SUBAPPLICATION Uebung_080e2_AX (* Beispiel für E_CTU mit Eventbremse durch AX_D_FF / AUI_D_FF_TMIN *)
  (* Standard: 61499-2; Description: Copyright (c) 2023 Meisterschulen am Ostbahnhof This program and the accompanying materials are made available under the terms of the Eclipse Public License 2.0 which is available at https://www.eclipse.org/legal/epl-2.0/ SPDX-License-Identifier: EPL-2.0 *)
  (* Version 1.1, 2026-05-15, Franz Höpfinger, Meisterschulen am Ostbahnhof, Ported to AX Welt *)
  PACKAGE Uebungen;
  IMPORT logiBUS::io::DI::logiBUS_DI::Input_I1;
  IMPORT logiBUS::io::DI::logiBUS_DI::Input_I2;
  IMPORT logiBUS::io::DQ::logiBUS_DO::Output_Q1;
  IMPORT Uebungen::const::UT::DefaultPool::OutputNumber_N1;
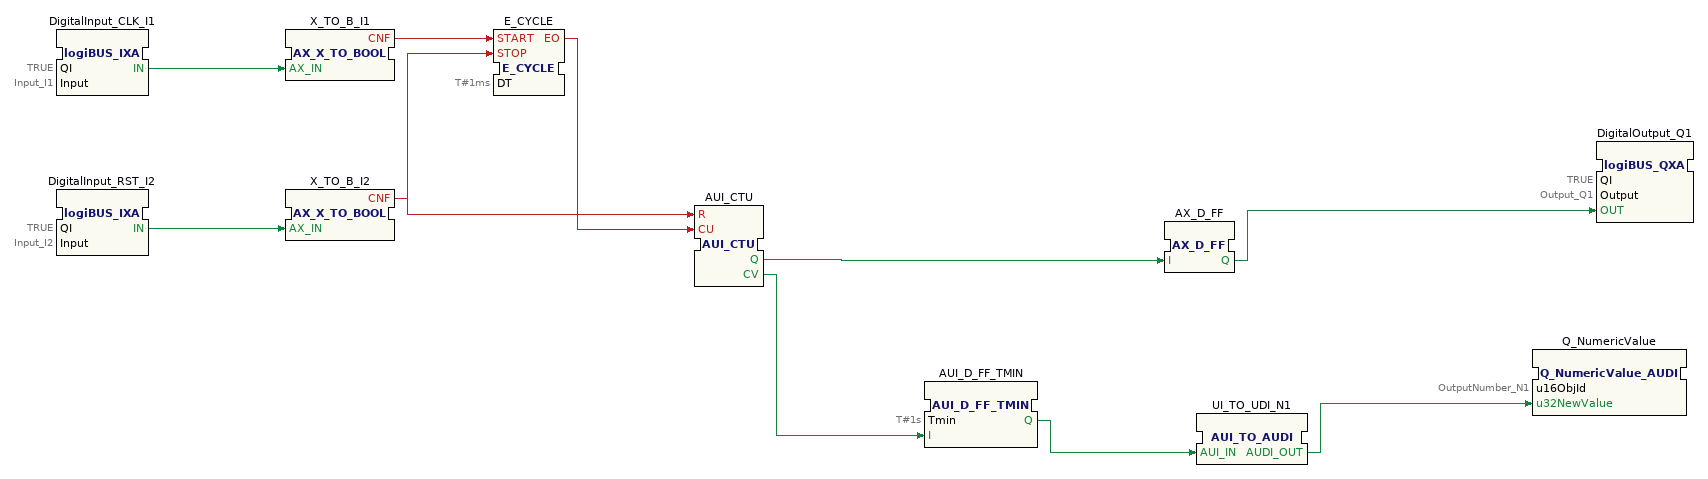
  FBS
    DigitalOutput_Q1 : logiBUS::io::DQ::logiBUS_QXA(QI := TRUE, Output := Output_Q1);
    DigitalInput_CLK_I1 : logiBUS::io::DI::logiBUS_IXA(QI := TRUE, Input := Input_I1);
    AUI_CTU : adapter::events::unidirectional::AUI_CTU;
    DigitalInput_RST_I2 : logiBUS::io::DI::logiBUS_IXA(QI := TRUE, Input := Input_I2);
    AX_D_FF : adapter::events::unidirectional::AX_D_FF;
    AUI_D_FF_TMIN : adapter::events::unidirectional::AUI_D_FF_TMIN(Tmin := T#1s);
    Q_NumericValue : isobus::UT::Q::Q_NumericValue_AUDI(u16ObjId := OutputNumber_N1);
    E_CYCLE : iec61499::events::E_CYCLE(DT := T#1ms);
    X_TO_B_I1 : adapter::conversion::unidirectional::AX_X_TO_BOOL;
    X_TO_B_I2 : adapter::conversion::unidirectional::AX_X_TO_BOOL;
    UI_TO_UDI_N1 : adapter::conversion::unidirectional::AUI_TO_AUDI;
  END_FBS
  EVENT_CONNECTIONS
    X_TO_B_I1.CNF TO E_CYCLE.START;
    X_TO_B_I2.CNF TO AUI_CTU.R;
    X_TO_B_I2.CNF TO E_CYCLE.STOP;
    E_CYCLE.EO TO AUI_CTU.CU;
  END_CONNECTIONS
  ADAPTER_CONNECTIONS
    DigitalInput_CLK_I1.IN TO X_TO_B_I1.AX_IN;
    DigitalInput_RST_I2.IN TO X_TO_B_I2.AX_IN;
    AX_D_FF.Q TO DigitalOutput_Q1.OUT;
    AUI_D_FF_TMIN.Q TO UI_TO_UDI_N1.AUI_IN;
    UI_TO_UDI_N1.AUDI_OUT TO Q_NumericValue.u32NewValue;
    AUI_CTU.Q TO AX_D_FF.I;
    AUI_CTU.CV TO AUI_D_FF_TMIN.I;
  END_CONNECTIONS
END_SUBAPPLICATION
